// Output from safety check task
// Input to master arm control task
TYPE ST_SafetyData :
STRUCT
	m_faultTrigged:BOOL := FALSE;
END_STRUCT
END_TYPE

(* stored: Version 1.1.0.1, ProductVersion 3.1.4024.12
   DUT ST_SafetyData: Id {322b279b-f9a5-4da8-8f90-8d4b82ec3137} *)
